(* Logix 5000 project; controller LeakTestAuto vendor 1 type 14 code 226 rev 37.11; software revision 37.01; part 5 of 12 *)
(* tags used below, declared in another part *)
   AOI_CTS1 : AOI_CTS_INSTRUMENT;
   AOI_CTS2 : AOI_CTS_INSTRUMENT;
   AOI_OP220_HomingSeq : AOI_Sequencer_x64;
   AOI_RobotPos : AOI_RobotPositions;
   AOI_SeqSteps : AOI_StandardSeqSteps;
   BarcodeScanner : udt_OutputStructure;
   Config_ConveyorHomeCounter : DINT;
   Config_ConveyorHomeCounterEnter : BOOL;
   Config_CylinderWaitTime : DINT;
   Config_CylinderWaitTimeEnter : BOOL;
   Config_MaxFailCount : DINT;
   Config_MaxFailCountEnter : BOOL;
   Conveyor : udt_OutputStructure;
   Conveyor_Seq : udt_SequenceStructure_X64;
   ConveyorHomeCounter : COUNTER;
   DryCycle_N1Ready : BOOL;
   DryCycle_N2Ready : BOOL;
   FailCount : COUNTER;
   HMI_CloseDisplay : DINT;
   HomingClearNestsBypass : BOOL;
   LeakTester1 : udt_OutputStructure;
   LeakTester2 : udt_OutputStructure;
   Mode_CapActuators : BOOL;
   Mode_CapCTS : BOOL;
   Mode_CapCylinders : BOOL;
   Mode_CapFail : BOOL;
   Mode_CapPass : BOOL;
   Mode_CapRobot : BOOL;
   Mode_CapShuffle : BOOL;
   Nest1Cylinder : udt_OutputStructure;
   Nest1Empty : BOOL;
   Nest1Ready : BOOL;
   Nest2Cylinder : udt_OutputStructure;
   Nest2Empty : BOOL;
   Nest2Ready : BOOL;
   ONS_CycleStop : BOOL;
   ONS_FailBinRemoved : BOOL;
   ONS_ManuMode : BOOL;
   OP220 : udt_Mode;
   OP220_HomingSeq : udt_SequenceStructure_X64;
   OP220_PartToPartCycleTMR : TIMER;
   OP220_Seq : udt_SequenceStructure_X64;
   RFIDScanner : udt_OutputStructure;
   Robot : udt_OutputStructure;
   RobotGripper : udt_OutputStructure;
   RobotInputs : udt_EpsonInputs;
   RobotOutputs : udt_EpsonOutputs;
   TON_FailChute : TIMER[10];
   TON_HMICloseDisplayDelay : TIMER;
   TON_Nest1DryCycleDryTest : TIMER;
   TON_Nest2DryCycleDryTest : TIMER;
   ConveyorPurgeCounter : DINT;   // Outfeed Coveyor Purge Counter
   HMI_PurgeCycleSP : DINT;   // HMI Purge Cycles Setpoint
   I_OP220_N3_CONVEYOR_CLEAT : ALIAS FOR Local:3:I.Pt13.Data;
   I_OP220_N3_DUT_PRE_NEST_1 : ALIAS FOR Local:3:I.Pt01.Data;
   I_OP220_N3_DUT_PRE_NEST_2 : ALIAS FOR Local:3:I.Pt02.Data;
   I_OP220_N3_MAIN_AIR_OK : ALIAS FOR Local:3:I.Pt07.Data;
   I_OP220_N3_NEST1_EXTEND : ALIAS FOR Local:3:I.Pt04.Data;
   I_OP220_N3_NEST1_HOME : ALIAS FOR Local:3:I.Pt03.Data;
   I_OP220_N3_NEST2_EXTEND : ALIAS FOR Local:3:I.Pt06.Data;
   I_OP220_N3_NEST2_HOME : ALIAS FOR Local:3:I.Pt05.Data;
   I_OP220_N3_REJECT_BIN_OK : ALIAS FOR Local:3:I.Pt09.Data;
   I_OP220_N3_REJECT_CHUTE_PART : ALIAS FOR Local:3:I.Pt10.Data;
   James_Dint : DINT;   // James Test Word
   O_OP220_N5_CONV_REV : ALIAS FOR Local:5:O.Pt11.Data;
   O_OP220_N5_EN_LT_BU : ALIAS FOR Local:5:O.Pt03.Data;
   O_OP220_N5_EN_LT_GN : ALIAS FOR Local:5:O.Pt00.Data;
   O_OP220_N5_EN_LT_RD : ALIAS FOR Local:5:O.Pt02.Data;
   O_OP220_N5_EN_LT_YE : ALIAS FOR Local:5:O.Pt01.Data;
   O_OP220_N5_EN_MAIN_AIR : ALIAS FOR Local:5:O.Pt04.Data;
   O_OP220_N5_EN_ROBOT_LATCHOFF : ALIAS FOR Local:5:O.Pt09.Data;
   OP220_ConsumedFromMain_PurgeModeEn : BOOL;
   OP220_Power : BOOL;
   PLC : AOI_PLC;
   Purge_Count_DN : BOOL;   // Purge Counter Completed
(* MainProgram, continued *)

ROUTINE R05_ModeControl   (* ladder *)
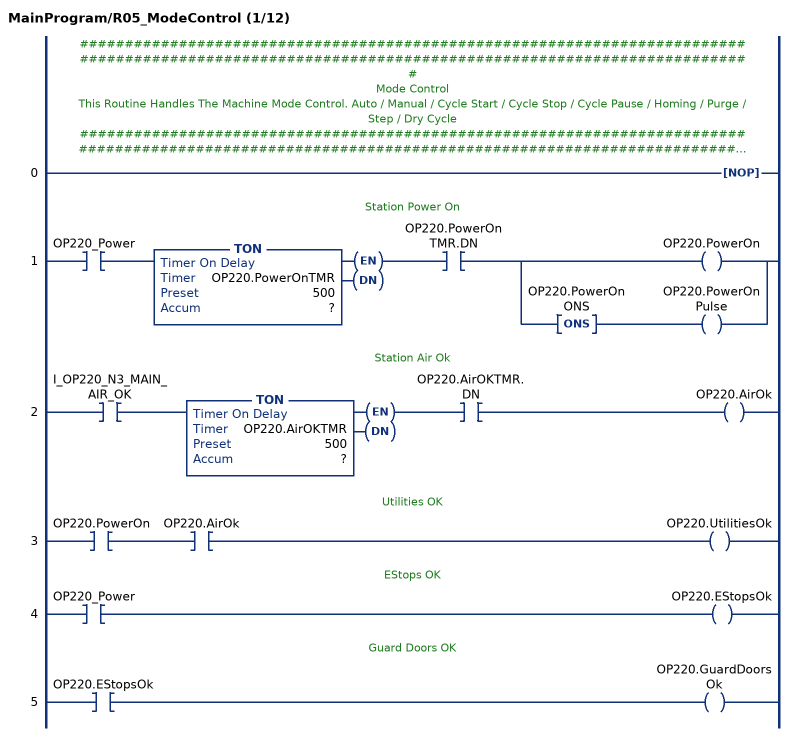
   // #####################################################################################################################################################
   // Mode Control
   // This Routine Handles The Machine Mode Control. Auto / Manual / Cycle Start / Cycle Stop / Cycle Pause / Homing / Purge / Step / Dry Cycle
   // #####################################################################################################################################################
   0: NOP();
   // Station Power On
   1: XIC(OP220_Power)TON(OP220.PowerOnTMR,?,?)XIC(OP220.PowerOnTMR.DN)[OTE(OP220.PowerOn) ,ONS(OP220.PowerOnONS) OTE(OP220.PowerOnPulse) ];
   // Station Air Ok
   2: XIC(I_OP220_N3_MAIN_AIR_OK)TON(OP220.AirOKTMR,?,?)XIC(OP220.AirOKTMR.DN)OTE(OP220.AirOk);
   // Utilities OK
   3: XIC(OP220.PowerOn)XIC(OP220.AirOk)OTE(OP220.UtilitiesOk);
   // EStops OK
   4: XIC(OP220_Power)OTE(OP220.EStopsOk);
   // Guard Doors OK
   5: XIC(OP220.EStopsOk)OTE(OP220.GuardDoorsOk);
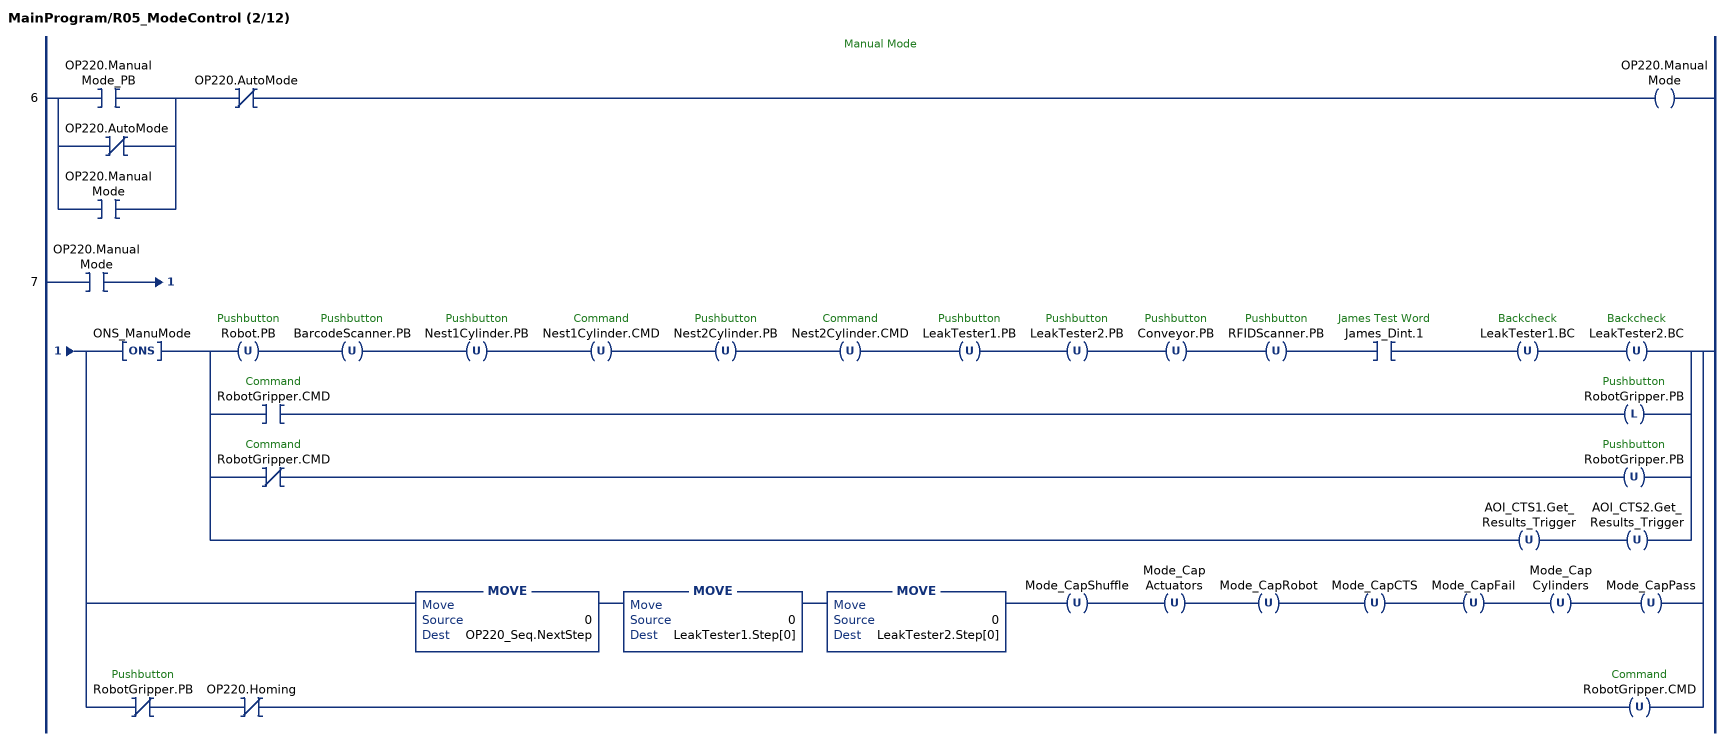
   // Manual Mode
   6: [XIC(OP220.ManualMode_PB) ,XIO(OP220.AutoMode) ,XIC(OP220.ManualMode) ]XIO(OP220.AutoMode)OTE(OP220.ManualMode);
   7: XIC(OP220.ManualMode)[ONS(ONS_ManuMode) [OTU(Robot.PB) OTU(BarcodeScanner.PB) OTU(Nest1Cylinder.PB) OTU(Nest1Cylinder.CMD) OTU(Nest2Cylinder.PB) OTU(Nest2Cylinder.CMD) OTU(LeakTester1.PB) OTU(LeakTester2.PB) OTU(Conveyor.PB) OTU(RFIDScanner.PB) XIC(James_Dint.1) OTU(LeakTester1.BC) OTU(LeakTester2.BC) ,XIC(RobotGripper.CMD) OTL(RobotGripper.PB) ,XIO(RobotGripper.CMD) OTU(RobotGripper.PB) ,OTU(AOI_CTS1.Get_Results_Trigger) OTU(AOI_CTS2.Get_Results_Trigger) ] ,MOVE(0,OP220_Seq.NextStep) MOVE(0,LeakTester1.Step[0]) MOVE(0,LeakTester2.Step[0]) OTU(Mode_CapShuffle) OTU(Mode_CapActuators) OTU(Mode_CapRobot) OTU(Mode_CapCTS) OTU(Mode_CapFail) OTU(Mode_CapCylinders) OTU(Mode_CapPass) ,XIO(RobotGripper.PB) XIO(OP220.Homing) OTU(RobotGripper.CMD) ];
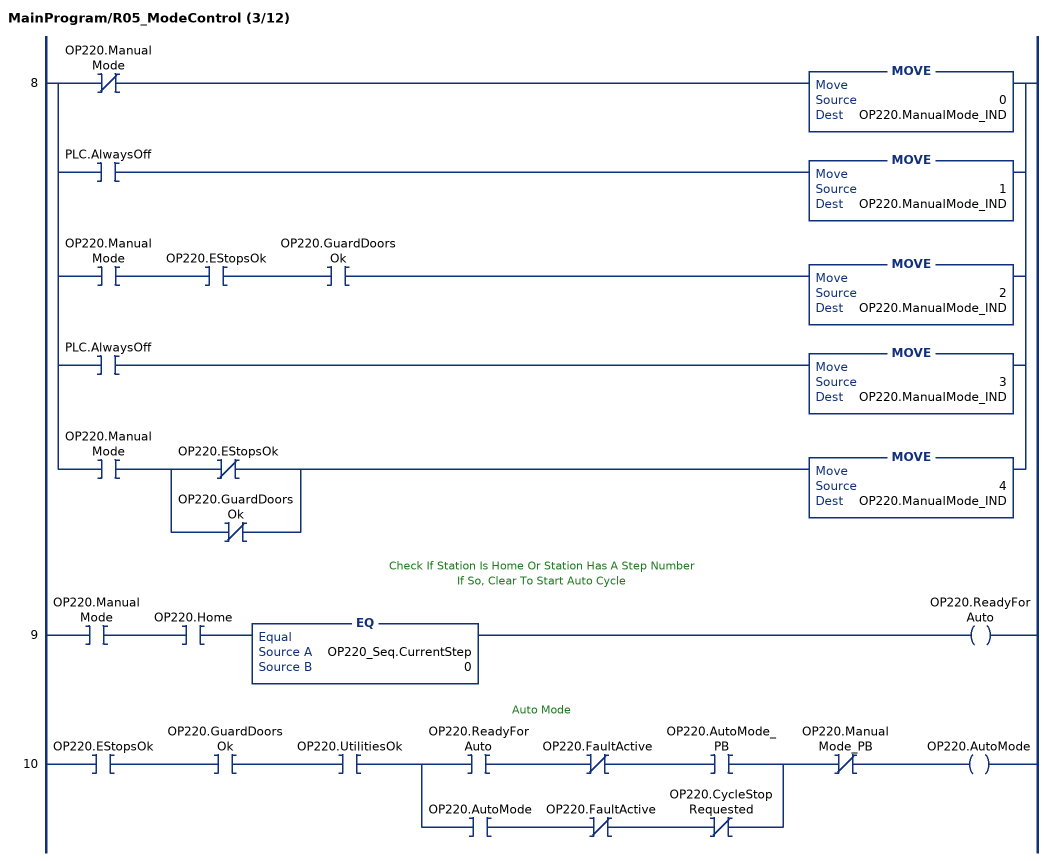
   8: [XIO(OP220.ManualMode) MOVE(0,OP220.ManualMode_IND) ,XIC(PLC.AlwaysOff) MOVE(1,OP220.ManualMode_IND) ,XIC(OP220.ManualMode) XIC(OP220.EStopsOk) XIC(OP220.GuardDoorsOk) MOVE(2,OP220.ManualMode_IND) ,XIC(PLC.AlwaysOff) MOVE(3,OP220.ManualMode_IND) ,XIC(OP220.ManualMode) [XIO(OP220.EStopsOk) ,XIO(OP220.GuardDoorsOk) ] MOVE(4,OP220.ManualMode_IND) ];
   // Check If Station Is Home Or Station Has A Step Number
   // If So, Clear To Start Auto Cycle
   9: XIC(OP220.ManualMode)XIC(OP220.Home)EQ(OP220_Seq.CurrentStep,0)OTE(OP220.ReadyForAuto);
   // Auto Mode
   10: XIC(OP220.EStopsOk)XIC(OP220.GuardDoorsOk)XIC(OP220.UtilitiesOk)[XIC(OP220.ReadyForAuto) XIO(OP220.FaultActive) XIC(OP220.AutoMode_PB) ,XIC(OP220.AutoMode) XIO(OP220.FaultActive) XIO(OP220.CycleStopRequested) ]XIO(OP220.ManualMode_PB)OTE(OP220.AutoMode);
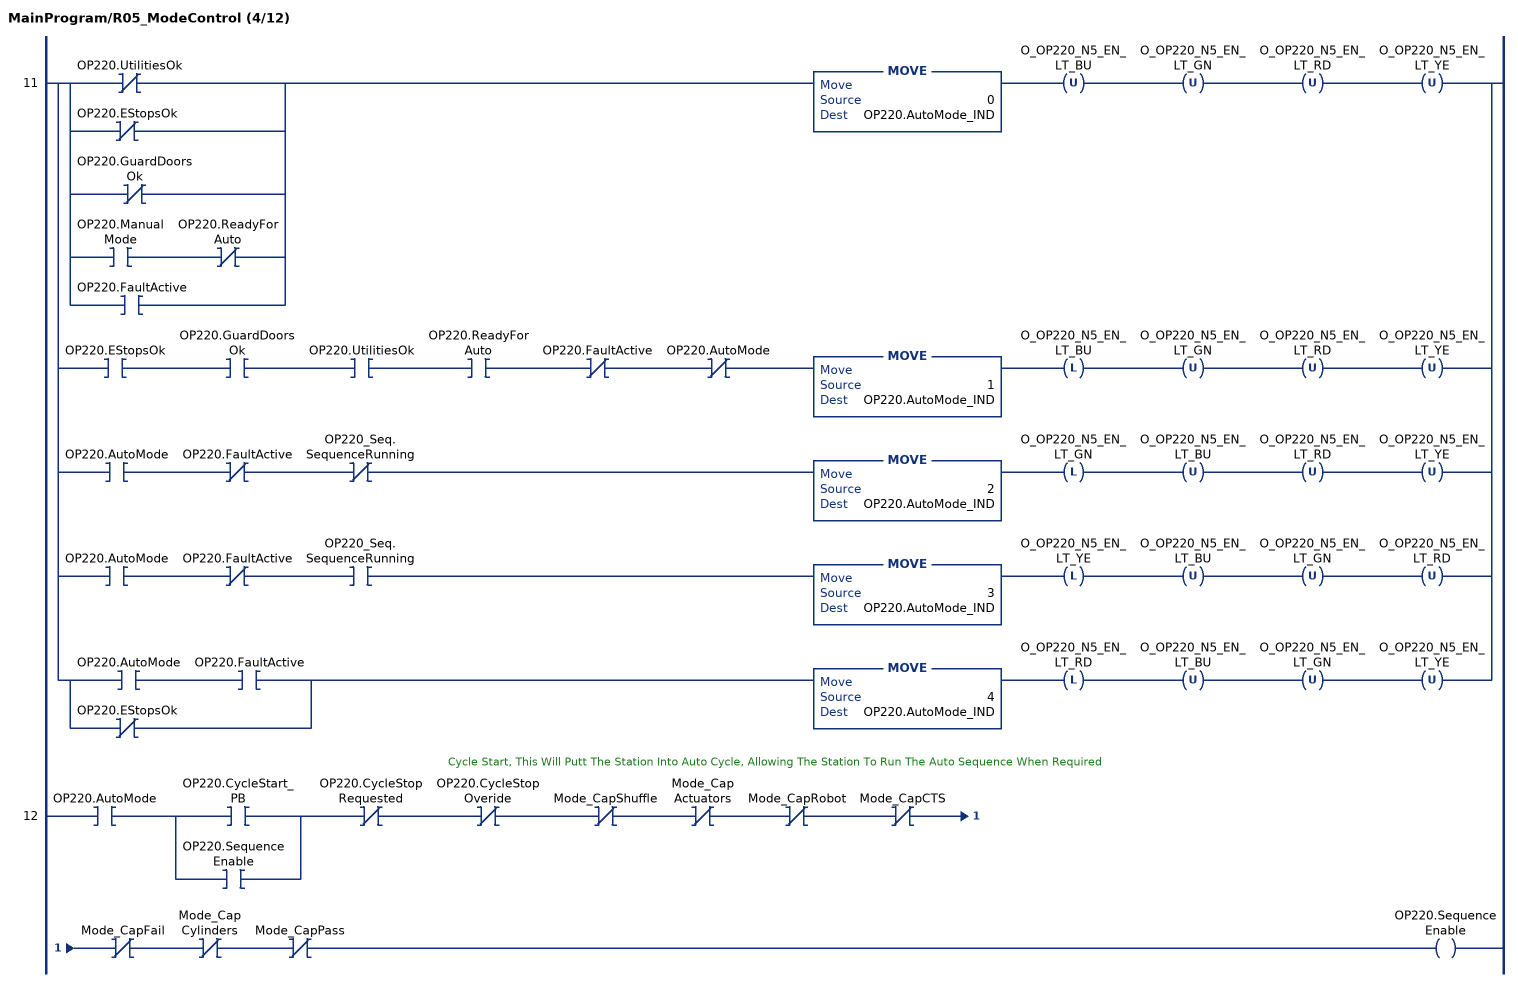
   11: [[XIO(OP220.UtilitiesOk) ,XIO(OP220.EStopsOk) ,XIO(OP220.GuardDoorsOk) ,XIC(OP220.ManualMode) XIO(OP220.ReadyForAuto) ,XIC(OP220.FaultActive) ] MOVE(0,OP220.AutoMode_IND) OTU(O_OP220_N5_EN_LT_BU) OTU(O_OP220_N5_EN_LT_GN) OTU(O_OP220_N5_EN_LT_RD) OTU(O_OP220_N5_EN_LT_YE) ,XIC(OP220.EStopsOk) XIC(OP220.GuardDoorsOk) XIC(OP220.UtilitiesOk) XIC(OP220.ReadyForAuto) XIO(OP220.FaultActive) XIO(OP220.AutoMode) MOVE(1,OP220.AutoMode_IND) OTL(O_OP220_N5_EN_LT_BU) OTU(O_OP220_N5_EN_LT_GN) OTU(O_OP220_N5_EN_LT_RD) OTU(O_OP220_N5_EN_LT_YE) ,XIC(OP220.AutoMode) XIO(OP220.FaultActive) XIO(OP220_Seq.SequenceRunning) MOVE(2,OP220.AutoMode_IND) OTL(O_OP220_N5_EN_LT_GN) OTU(O_OP220_N5_EN_LT_BU) OTU(O_OP220_N5_EN_LT_RD) OTU(O_OP220_N5_EN_LT_YE) ,XIC(OP220.AutoMode) XIO(OP220.FaultActive) XIC(OP220_Seq.SequenceRunning) MOVE(3,OP220.AutoMode_IND) OTL(O_OP220_N5_EN_LT_YE) OTU(O_OP220_N5_EN_LT_BU) OTU(O_OP220_N5_EN_LT_GN) OTU(O_OP220_N5_EN_LT_RD) ,[XIC(OP220.AutoMode) XIC(OP220.FaultActive) ,XIO(OP220.EStopsOk) ] MOVE(4,OP220.AutoMode_IND) OTL(O_OP220_N5_EN_LT_RD) OTU(O_OP220_N5_EN_LT_BU) OTU(O_OP220_N5_EN_LT_GN) OTU(O_OP220_N5_EN_LT_YE) ];
   // Cycle Start, This Will Putt The Station Into Auto Cycle, Allowing The Station To Run The Auto Sequence When Required
   12: XIC(OP220.AutoMode)[XIC(OP220.CycleStart_PB) ,XIC(OP220.SequenceEnable) ]XIO(OP220.CycleStopRequested)XIO(OP220.CycleStopOveride)XIO(Mode_CapShuffle)XIO(Mode_CapActuators)XIO(Mode_CapRobot)XIO(Mode_CapCTS)XIO(Mode_CapFail)XIO(Mode_CapCylinders)XIO(Mode_CapPass)OTE(OP220.SequenceEnable);
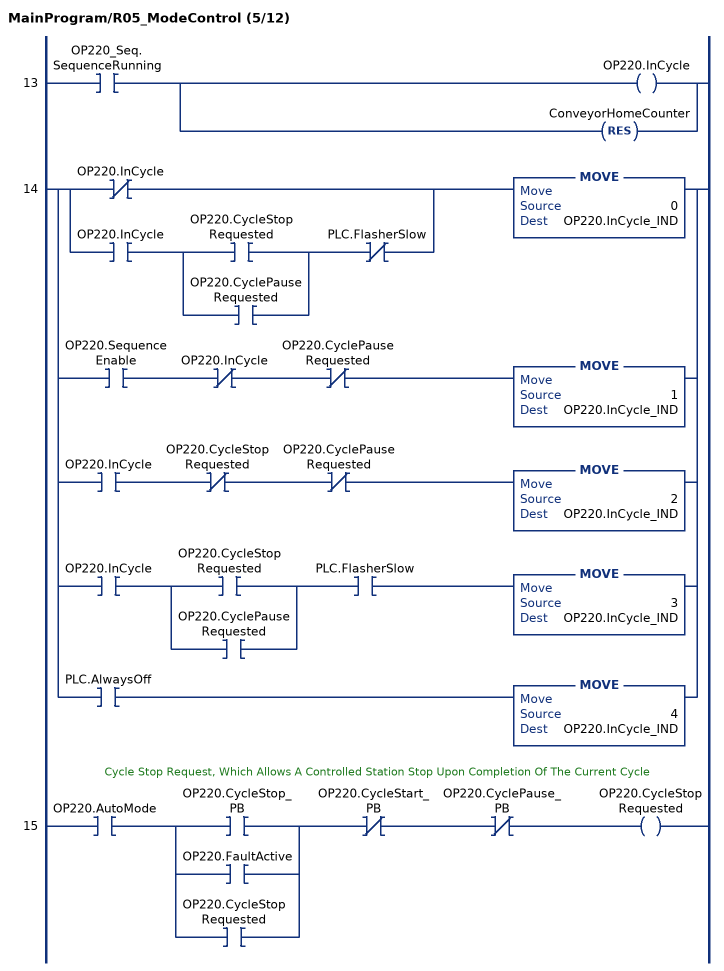
   13: XIC(OP220_Seq.SequenceRunning)[OTE(OP220.InCycle) ,RES(ConveyorHomeCounter) ];
   14: [[XIO(OP220.InCycle) ,XIC(OP220.InCycle) [XIC(OP220.CycleStopRequested) ,XIC(OP220.CyclePauseRequested) ] XIO(PLC.FlasherSlow) ] MOVE(0,OP220.InCycle_IND) ,XIC(OP220.SequenceEnable) XIO(OP220.InCycle) XIO(OP220.CyclePauseRequested) MOVE(1,OP220.InCycle_IND) ,XIC(OP220.InCycle) XIO(OP220.CycleStopRequested) XIO(OP220.CyclePauseRequested) MOVE(2,OP220.InCycle_IND) ,XIC(OP220.InCycle) [XIC(OP220.CycleStopRequested) ,XIC(OP220.CyclePauseRequested) ] XIC(PLC.FlasherSlow) MOVE(3,OP220.InCycle_IND) ,XIC(PLC.AlwaysOff) MOVE(4,OP220.InCycle_IND) ];
   // Cycle Stop Request, Which Allows A Controlled Station Stop Upon Completion Of The Current Cycle
   15: XIC(OP220.AutoMode)[XIC(OP220.CycleStop_PB) ,XIC(OP220.FaultActive) ,XIC(OP220.CycleStopRequested) ]XIO(OP220.CycleStart_PB)XIO(OP220.CyclePause_PB)OTE(OP220.CycleStopRequested);
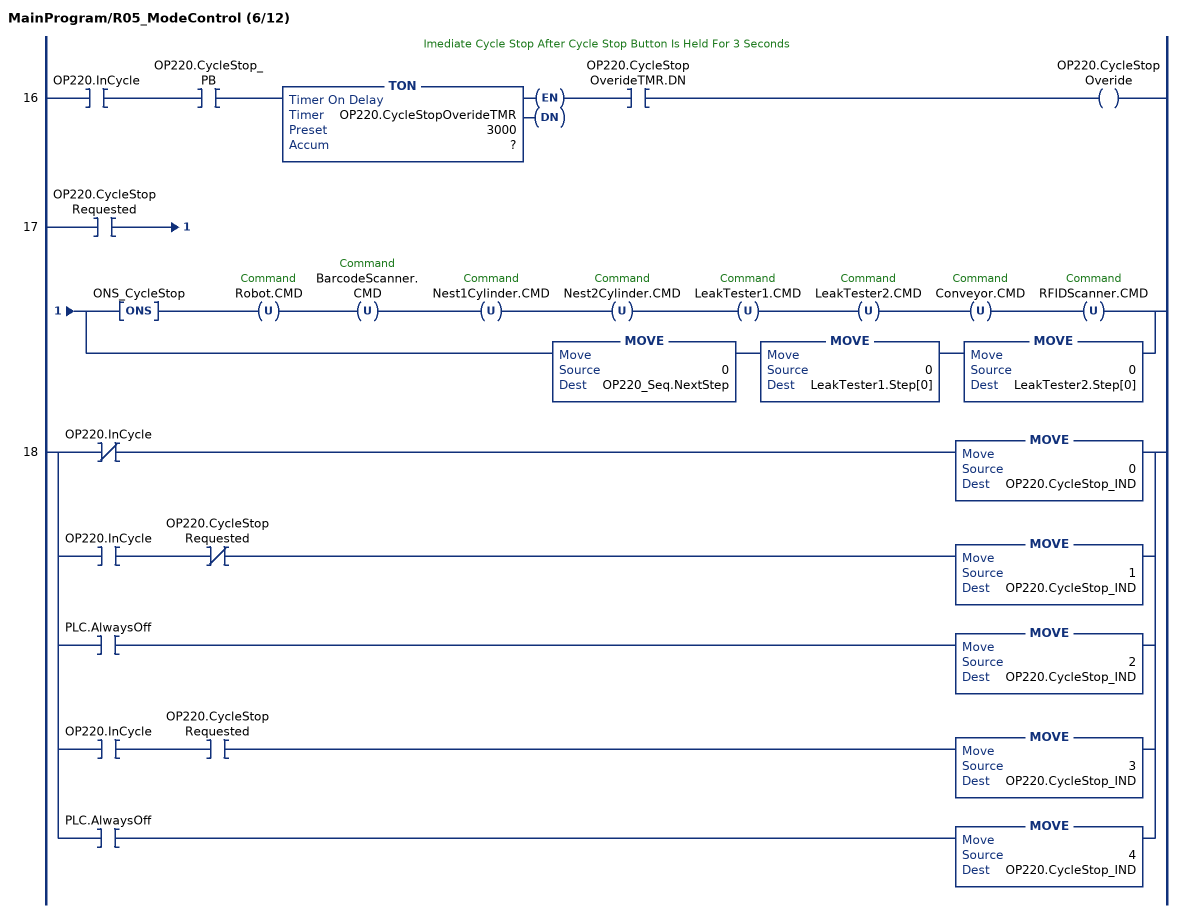
   // Imediate Cycle Stop After Cycle Stop Button Is Held For 3 Seconds
   16: XIC(OP220.InCycle)XIC(OP220.CycleStop_PB)TON(OP220.CycleStopOverideTMR,?,?)XIC(OP220.CycleStopOverideTMR.DN)OTE(OP220.CycleStopOveride);
   17: XIC(OP220.CycleStopRequested)[ONS(ONS_CycleStop) OTU(Robot.CMD) OTU(BarcodeScanner.CMD) OTU(Nest1Cylinder.CMD) OTU(Nest2Cylinder.CMD) OTU(LeakTester1.CMD) OTU(LeakTester2.CMD) OTU(Conveyor.CMD) OTU(RFIDScanner.CMD) ,MOVE(0,OP220_Seq.NextStep) MOVE(0,LeakTester1.Step[0]) MOVE(0,LeakTester2.Step[0]) ];
   18: [XIO(OP220.InCycle) MOVE(0,OP220.CycleStop_IND) ,XIC(OP220.InCycle) XIO(OP220.CycleStopRequested) MOVE(1,OP220.CycleStop_IND) ,XIC(PLC.AlwaysOff) MOVE(2,OP220.CycleStop_IND) ,XIC(OP220.InCycle) XIC(OP220.CycleStopRequested) MOVE(3,OP220.CycleStop_IND) ,XIC(PLC.AlwaysOff) MOVE(4,OP220.CycleStop_IND) ];
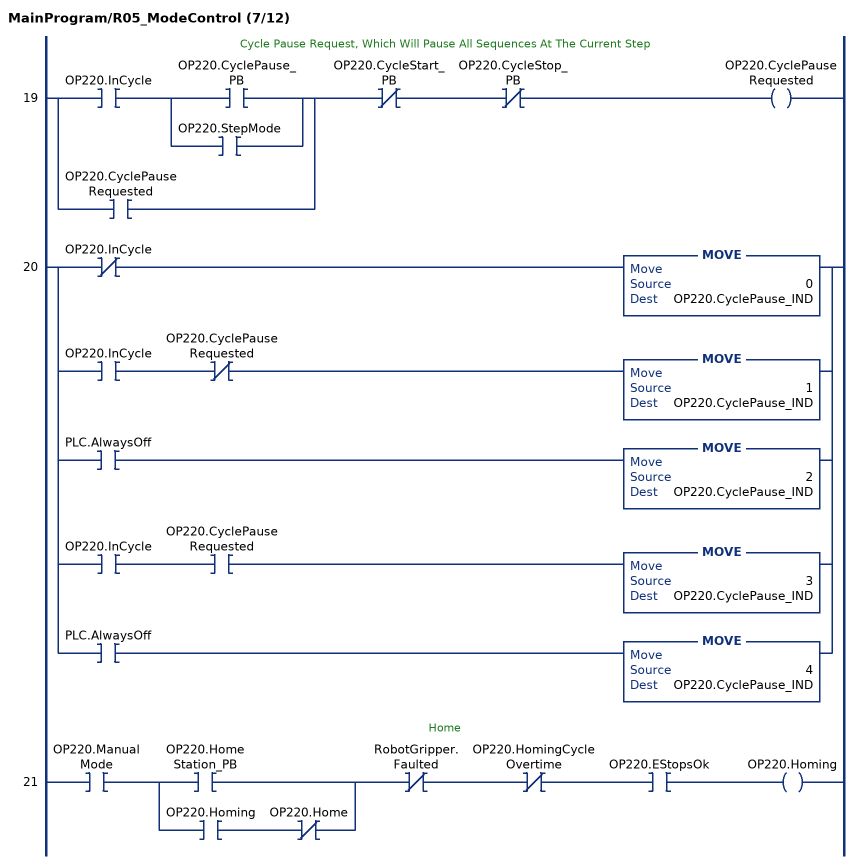
   // Cycle Pause Request, Which Will Pause All Sequences At The Current Step
   19: [XIC(OP220.InCycle) [XIC(OP220.CyclePause_PB) ,XIC(OP220.StepMode) ] ,XIC(OP220.CyclePauseRequested) ]XIO(OP220.CycleStart_PB)XIO(OP220.CycleStop_PB)OTE(OP220.CyclePauseRequested);
   20: [XIO(OP220.InCycle) MOVE(0,OP220.CyclePause_IND) ,XIC(OP220.InCycle) XIO(OP220.CyclePauseRequested) MOVE(1,OP220.CyclePause_IND) ,XIC(PLC.AlwaysOff) MOVE(2,OP220.CyclePause_IND) ,XIC(OP220.InCycle) XIC(OP220.CyclePauseRequested) MOVE(3,OP220.CyclePause_IND) ,XIC(PLC.AlwaysOff) MOVE(4,OP220.CyclePause_IND) ];
   // Home
   21: XIC(OP220.ManualMode)[XIC(OP220.HomeStation_PB) ,XIC(OP220.Homing) XIO(OP220.Home) ]XIO(RobotGripper.Faulted)XIO(OP220.HomingCycleOvertime)XIC(OP220.EStopsOk)OTE(OP220.Homing);
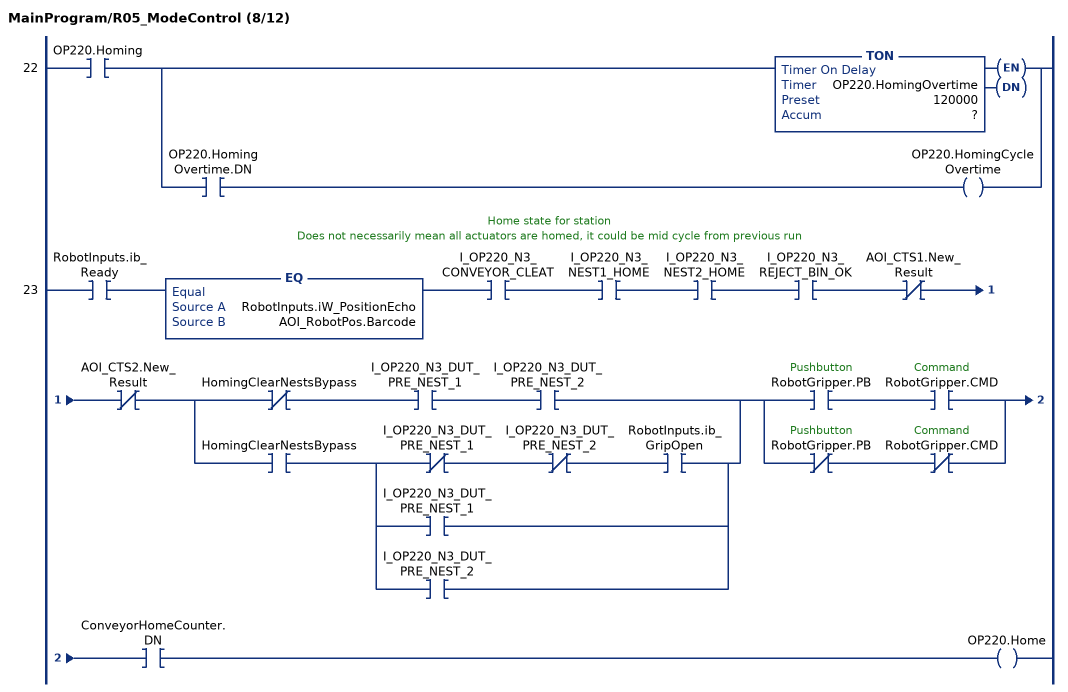
   22: XIC(OP220.Homing)[TON(OP220.HomingOvertime,?,?) ,XIC(OP220.HomingOvertime.DN) OTE(OP220.HomingCycleOvertime) ];
   // Home state for station
   // Does not necessarily mean all actuators are homed, it could be mid cycle from previous run
   23: XIC(RobotInputs.ib_Ready)EQ(RobotInputs.iW_PositionEcho,AOI_RobotPos.Barcode)XIC(I_OP220_N3_CONVEYOR_CLEAT)XIC(I_OP220_N3_NEST1_HOME)XIC(I_OP220_N3_NEST2_HOME)XIC(I_OP220_N3_REJECT_BIN_OK)XIO(AOI_CTS1.New_Result)XIO(AOI_CTS2.New_Result)[XIO(HomingClearNestsBypass) XIC(I_OP220_N3_DUT_PRE_NEST_1) XIC(I_OP220_N3_DUT_PRE_NEST_2) ,XIC(HomingClearNestsBypass) [XIO(I_OP220_N3_DUT_PRE_NEST_1) XIO(I_OP220_N3_DUT_PRE_NEST_2) XIC(RobotInputs.ib_GripOpen) ,XIC(I_OP220_N3_DUT_PRE_NEST_1) ,XIC(I_OP220_N3_DUT_PRE_NEST_2) ] ][XIC(RobotGripper.PB) XIC(RobotGripper.CMD) ,XIO(RobotGripper.PB) XIO(RobotGripper.CMD) ]XIC(ConveyorHomeCounter.DN)OTE(OP220.Home);
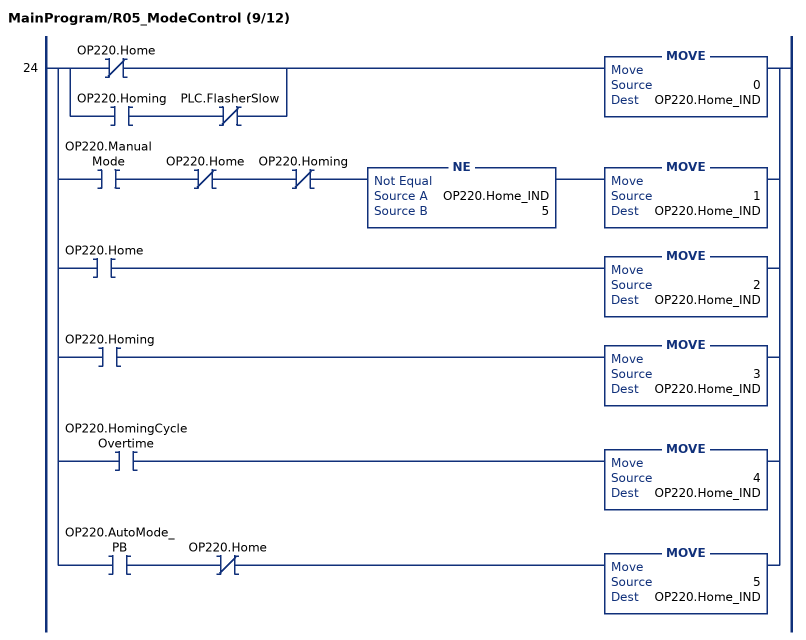
   24: [[XIO(OP220.Home) ,XIC(OP220.Homing) XIO(PLC.FlasherSlow) ] MOVE(0,OP220.Home_IND) ,XIC(OP220.ManualMode) XIO(OP220.Home) XIO(OP220.Homing) NE(OP220.Home_IND,5) MOVE(1,OP220.Home_IND) ,XIC(OP220.Home) MOVE(2,OP220.Home_IND) ,XIC(OP220.Homing) MOVE(3,OP220.Home_IND) ,XIC(OP220.HomingCycleOvertime) MOVE(4,OP220.Home_IND) ,XIC(OP220.AutoMode_PB) XIO(OP220.Home) MOVE(5,OP220.Home_IND) ];
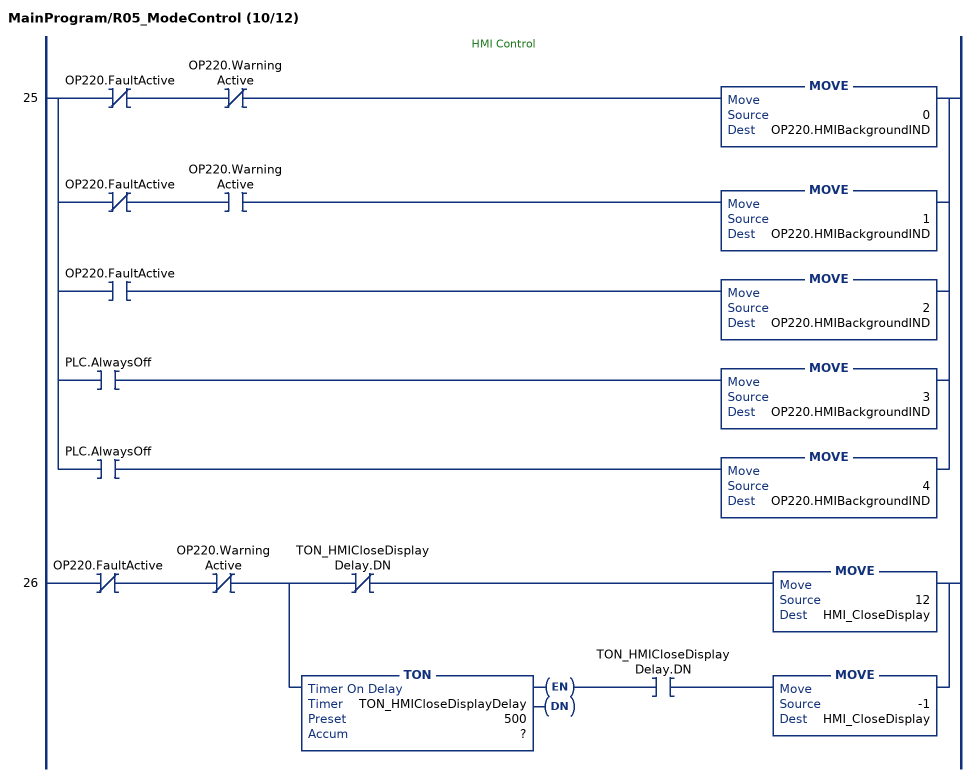
   // HMI Control
   25: [XIO(OP220.FaultActive) XIO(OP220.WarningActive) MOVE(0,OP220.HMIBackgroundIND) ,XIO(OP220.FaultActive) XIC(OP220.WarningActive) MOVE(1,OP220.HMIBackgroundIND) ,XIC(OP220.FaultActive) MOVE(2,OP220.HMIBackgroundIND) ,XIC(PLC.AlwaysOff) MOVE(3,OP220.HMIBackgroundIND) ,XIC(PLC.AlwaysOff) MOVE(4,OP220.HMIBackgroundIND) ];
   26: XIO(OP220.FaultActive)XIO(OP220.WarningActive)[XIO(TON_HMICloseDisplayDelay.DN) MOVE(12,HMI_CloseDisplay) ,TON(TON_HMICloseDisplayDelay,?,?) XIC(TON_HMICloseDisplayDelay.DN) MOVE(-1,HMI_CloseDisplay) ];
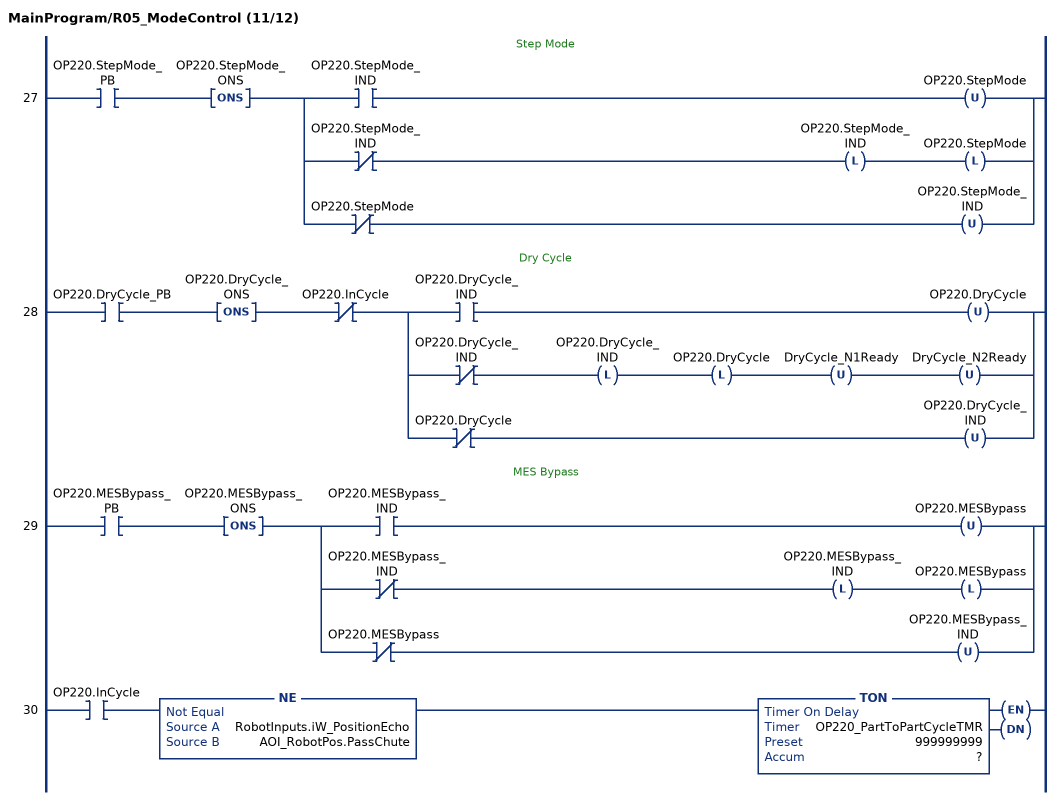
   // Step Mode
   27: XIC(OP220.StepMode_PB)ONS(OP220.StepMode_ONS)[XIC(OP220.StepMode_IND) OTU(OP220.StepMode) ,XIO(OP220.StepMode_IND) OTL(OP220.StepMode_IND) OTL(OP220.StepMode) ,XIO(OP220.StepMode) OTU(OP220.StepMode_IND) ];
   // Dry Cycle
   28: XIC(OP220.DryCycle_PB)ONS(OP220.DryCycle_ONS)XIO(OP220.InCycle)[XIC(OP220.DryCycle_IND) OTU(OP220.DryCycle) ,XIO(OP220.DryCycle_IND) OTL(OP220.DryCycle_IND) OTL(OP220.DryCycle) OTU(DryCycle_N1Ready) OTU(DryCycle_N2Ready) ,XIO(OP220.DryCycle) OTU(OP220.DryCycle_IND) ];
   // MES Bypass
   29: XIC(OP220.MESBypass_PB)ONS(OP220.MESBypass_ONS)[XIC(OP220.MESBypass_IND) OTU(OP220.MESBypass) ,XIO(OP220.MESBypass_IND) OTL(OP220.MESBypass_IND) OTL(OP220.MESBypass) ,XIO(OP220.MESBypass) OTU(OP220.MESBypass_IND) ];
   30: XIC(OP220.InCycle)NE(RobotInputs.iW_PositionEcho,AOI_RobotPos.PassChute)TON(OP220_PartToPartCycleTMR,?,?);
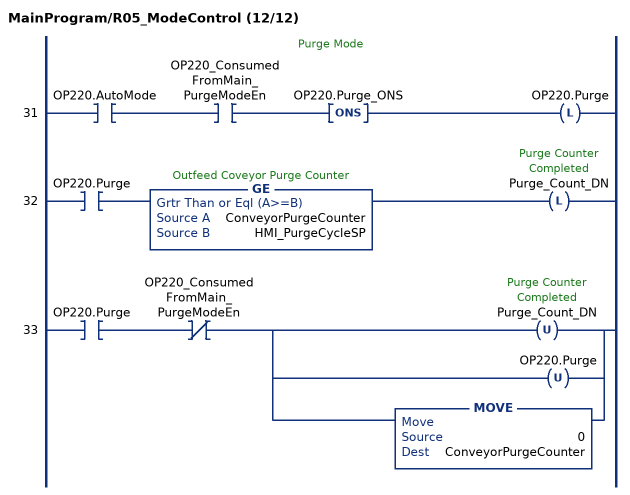
   // Purge Mode
   31: XIC(OP220.AutoMode)XIC(OP220_ConsumedFromMain_PurgeModeEn)ONS(OP220.Purge_ONS)OTL(OP220.Purge);
   32: XIC(OP220.Purge)GE(ConveyorPurgeCounter,HMI_PurgeCycleSP)OTL(Purge_Count_DN);
   33: XIC(OP220.Purge)XIO(OP220_ConsumedFromMain_PurgeModeEn)[OTU(Purge_Count_DN) ,OTU(OP220.Purge) ,MOVE(0,ConveyorPurgeCounter) ];
END_ROUTINE

ROUTINE R06_IOControl   (* ladder *)
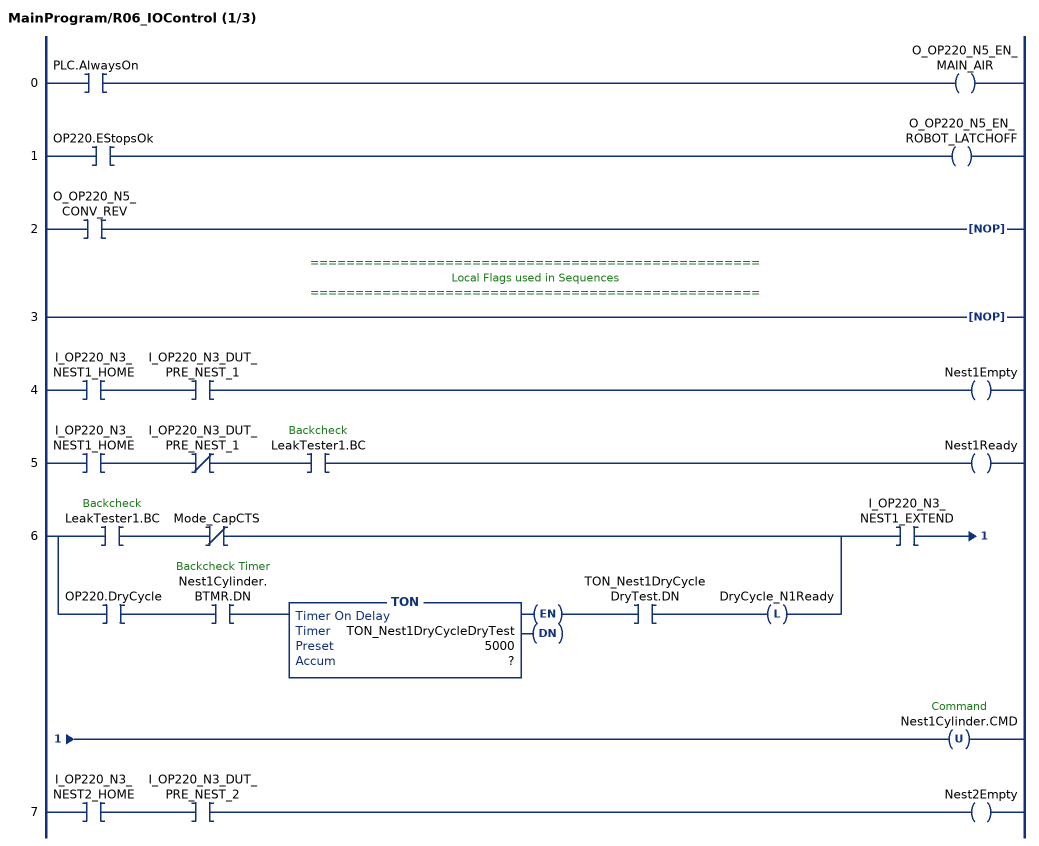
   0: XIC(PLC.AlwaysOn)OTE(O_OP220_N5_EN_MAIN_AIR);
   1: XIC(OP220.EStopsOk)OTE(O_OP220_N5_EN_ROBOT_LATCHOFF);
   2: XIC(O_OP220_N5_CONV_REV)NOP();
   // ==================================================
   // Local Flags used in Sequences
   // ==================================================
   3: NOP();
   4: XIC(I_OP220_N3_NEST1_HOME)XIC(I_OP220_N3_DUT_PRE_NEST_1)OTE(Nest1Empty);
   5: XIC(I_OP220_N3_NEST1_HOME)XIO(I_OP220_N3_DUT_PRE_NEST_1)XIC(LeakTester1.BC)OTE(Nest1Ready);
   6: [XIC(LeakTester1.BC) XIO(Mode_CapCTS) ,XIC(OP220.DryCycle) XIC(Nest1Cylinder.BTMR.DN) TON(TON_Nest1DryCycleDryTest,?,?) XIC(TON_Nest1DryCycleDryTest.DN) OTL(DryCycle_N1Ready) ]XIC(I_OP220_N3_NEST1_EXTEND)OTU(Nest1Cylinder.CMD);
   7: XIC(I_OP220_N3_NEST2_HOME)XIC(I_OP220_N3_DUT_PRE_NEST_2)OTE(Nest2Empty);
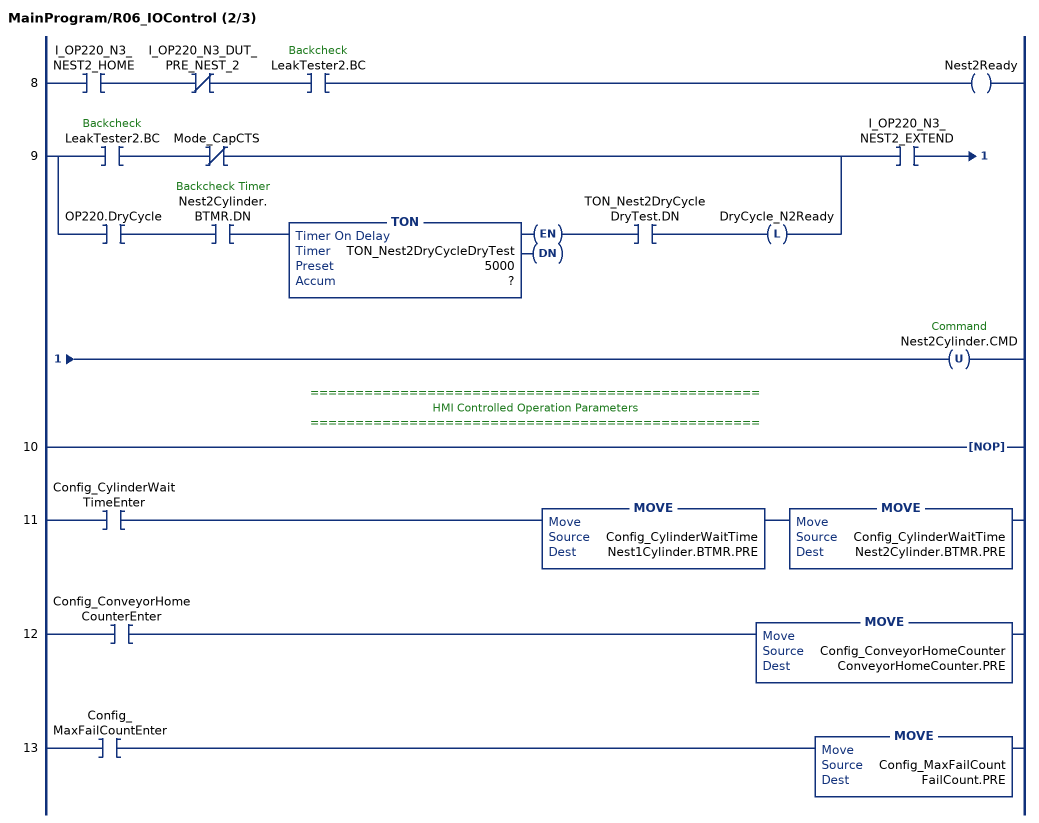
   8: XIC(I_OP220_N3_NEST2_HOME)XIO(I_OP220_N3_DUT_PRE_NEST_2)XIC(LeakTester2.BC)OTE(Nest2Ready);
   9: [XIC(LeakTester2.BC) XIO(Mode_CapCTS) ,XIC(OP220.DryCycle) XIC(Nest2Cylinder.BTMR.DN) TON(TON_Nest2DryCycleDryTest,?,?) XIC(TON_Nest2DryCycleDryTest.DN) OTL(DryCycle_N2Ready) ]XIC(I_OP220_N3_NEST2_EXTEND)OTU(Nest2Cylinder.CMD);
   // ==================================================
   // HMI Controlled Operation Parameters
   // ==================================================
   10: NOP();
   11: XIC(Config_CylinderWaitTimeEnter)MOVE(Config_CylinderWaitTime,Nest1Cylinder.BTMR.PRE)MOVE(Config_CylinderWaitTime,Nest2Cylinder.BTMR.PRE);
   12: XIC(Config_ConveyorHomeCounterEnter)MOVE(Config_ConveyorHomeCounter,ConveyorHomeCounter.PRE);
   13: XIC(Config_MaxFailCountEnter)MOVE(Config_MaxFailCount,FailCount.PRE);
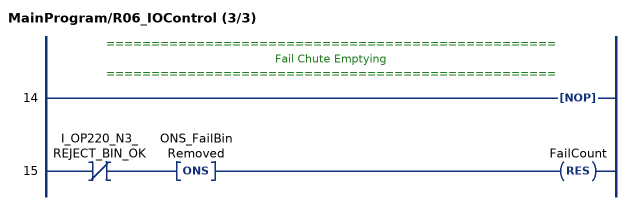
   // ==================================================
   // Fail Chute Emptying
   // ==================================================
   14: NOP();
   15: XIO(I_OP220_N3_REJECT_BIN_OK)ONS(ONS_FailBinRemoved)RES(FailCount);
END_ROUTINE

ROUTINE R09_Homing   (* ladder *)
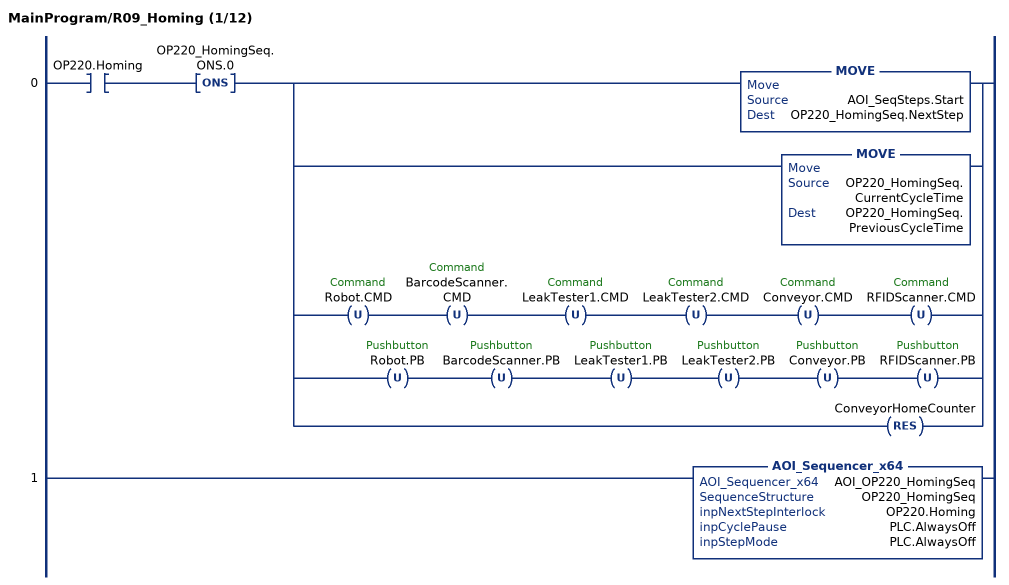
   0: XIC(OP220.Homing)ONS(OP220_HomingSeq.ONS.0)[MOVE(AOI_SeqSteps.Start,OP220_HomingSeq.NextStep) ,MOVE(OP220_HomingSeq.CurrentCycleTime,OP220_HomingSeq.PreviousCycleTime) ,OTU(Robot.CMD) OTU(BarcodeScanner.CMD) OTU(LeakTester1.CMD) OTU(LeakTester2.CMD) OTU(Conveyor.CMD) OTU(RFIDScanner.CMD) ,OTU(Robot.PB) OTU(BarcodeScanner.PB) OTU(LeakTester1.PB) OTU(LeakTester2.PB) OTU(Conveyor.PB) OTU(RFIDScanner.PB) ,RES(ConveyorHomeCounter) ];
   1: AOI_Sequencer_x64(AOI_OP220_HomingSeq,OP220_HomingSeq,OP220.Homing,PLC.AlwaysOff,PLC.AlwaysOff);
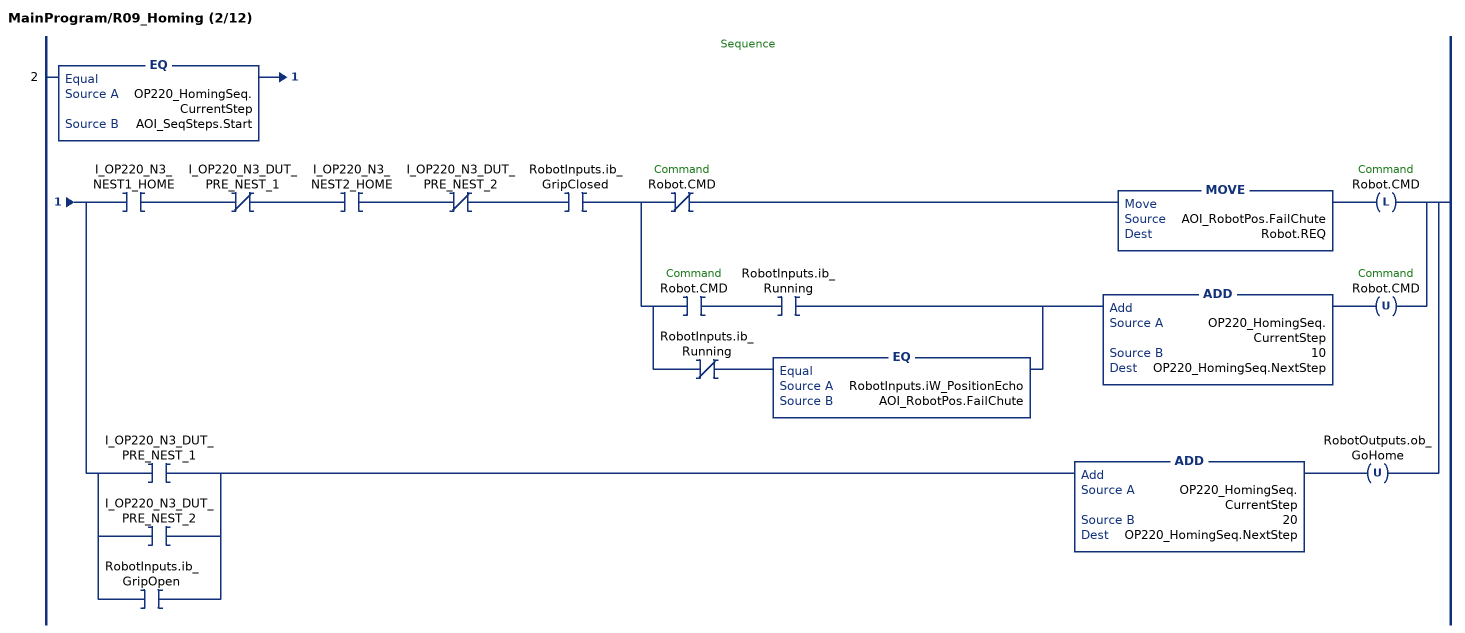
   // Sequence
   2: EQ(OP220_HomingSeq.CurrentStep,AOI_SeqSteps.Start)[XIC(I_OP220_N3_NEST1_HOME) XIO(I_OP220_N3_DUT_PRE_NEST_1) XIC(I_OP220_N3_NEST2_HOME) XIO(I_OP220_N3_DUT_PRE_NEST_2) XIC(RobotInputs.ib_GripClosed) [XIO(Robot.CMD) MOVE(AOI_RobotPos.FailChute,Robot.REQ) OTL(Robot.CMD) ,[XIC(Robot.CMD) XIC(RobotInputs.ib_Running) ,XIO(RobotInputs.ib_Running) EQ(RobotInputs.iW_PositionEcho,AOI_RobotPos.FailChute) ] ADD(OP220_HomingSeq.CurrentStep,10,OP220_HomingSeq.NextStep) OTU(Robot.CMD) ] ,[XIC(I_OP220_N3_DUT_PRE_NEST_1) ,XIC(I_OP220_N3_DUT_PRE_NEST_2) ,XIC(RobotInputs.ib_GripOpen) ] ADD(OP220_HomingSeq.CurrentStep,20,OP220_HomingSeq.NextStep) OTU(RobotOutputs.ob_GoHome) ];
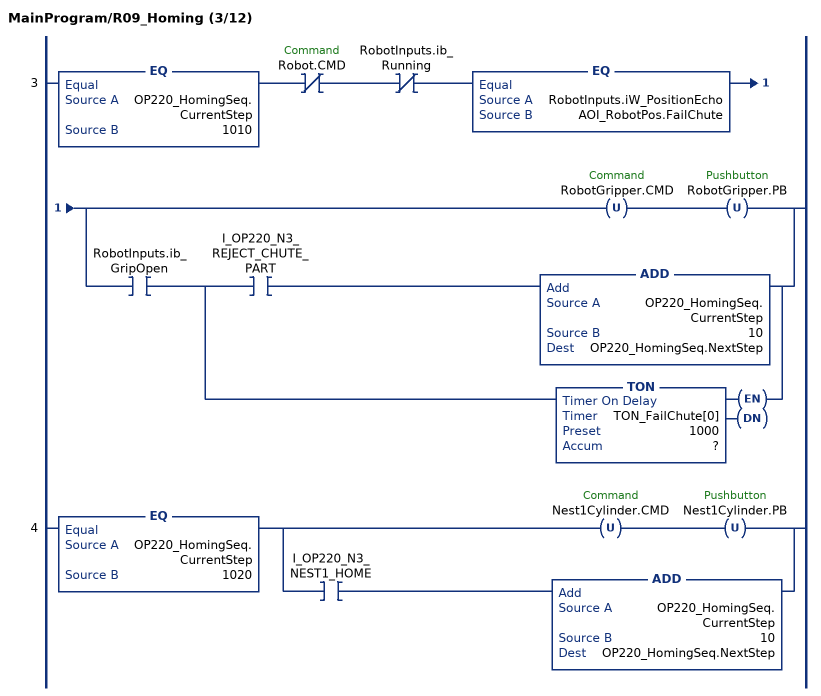
   3: EQ(OP220_HomingSeq.CurrentStep,1010)XIO(Robot.CMD)XIO(RobotInputs.ib_Running)EQ(RobotInputs.iW_PositionEcho,AOI_RobotPos.FailChute)[OTU(RobotGripper.CMD) OTU(RobotGripper.PB) ,XIC(RobotInputs.ib_GripOpen) [XIC(I_OP220_N3_REJECT_CHUTE_PART) ADD(OP220_HomingSeq.CurrentStep,10,OP220_HomingSeq.NextStep) ,TON(TON_FailChute[0],?,?) ] ];
   4: EQ(OP220_HomingSeq.CurrentStep,1020)[OTU(Nest1Cylinder.CMD) OTU(Nest1Cylinder.PB) ,XIC(I_OP220_N3_NEST1_HOME) ADD(OP220_HomingSeq.CurrentStep,10,OP220_HomingSeq.NextStep) ];
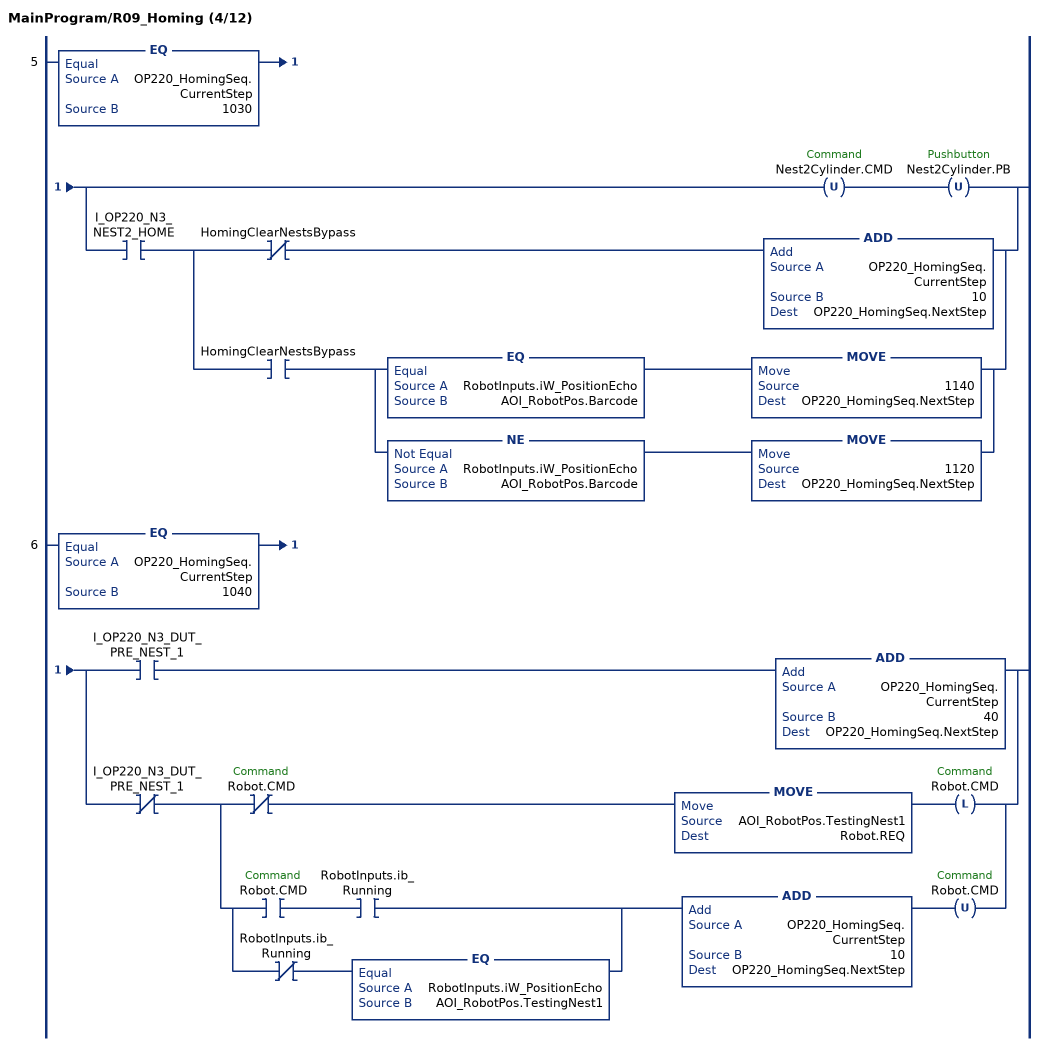
   5: EQ(OP220_HomingSeq.CurrentStep,1030)[OTU(Nest2Cylinder.CMD) OTU(Nest2Cylinder.PB) ,XIC(I_OP220_N3_NEST2_HOME) [XIO(HomingClearNestsBypass) ADD(OP220_HomingSeq.CurrentStep,10,OP220_HomingSeq.NextStep) ,XIC(HomingClearNestsBypass) [EQ(RobotInputs.iW_PositionEcho,AOI_RobotPos.Barcode) MOVE(1140,OP220_HomingSeq.NextStep) ,NE(RobotInputs.iW_PositionEcho,AOI_RobotPos.Barcode) MOVE(1120,OP220_HomingSeq.NextStep) ] ] ];
   6: EQ(OP220_HomingSeq.CurrentStep,1040)[XIC(I_OP220_N3_DUT_PRE_NEST_1) ADD(OP220_HomingSeq.CurrentStep,40,OP220_HomingSeq.NextStep) ,XIO(I_OP220_N3_DUT_PRE_NEST_1) [XIO(Robot.CMD) MOVE(AOI_RobotPos.TestingNest1,Robot.REQ) OTL(Robot.CMD) ,[XIC(Robot.CMD) XIC(RobotInputs.ib_Running) ,XIO(RobotInputs.ib_Running) EQ(RobotInputs.iW_PositionEcho,AOI_RobotPos.TestingNest1) ] ADD(OP220_HomingSeq.CurrentStep,10,OP220_HomingSeq.NextStep) OTU(Robot.CMD) ] ];
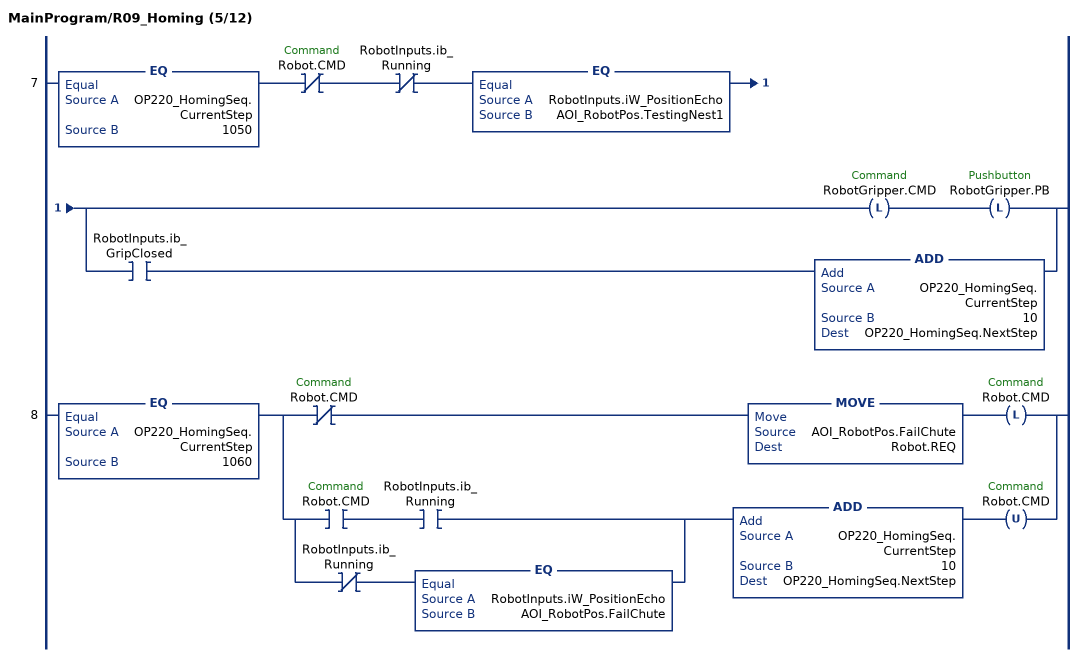
   7: EQ(OP220_HomingSeq.CurrentStep,1050)XIO(Robot.CMD)XIO(RobotInputs.ib_Running)EQ(RobotInputs.iW_PositionEcho,AOI_RobotPos.TestingNest1)[OTL(RobotGripper.CMD) OTL(RobotGripper.PB) ,XIC(RobotInputs.ib_GripClosed) ADD(OP220_HomingSeq.CurrentStep,10,OP220_HomingSeq.NextStep) ];
   8: EQ(OP220_HomingSeq.CurrentStep,1060)[XIO(Robot.CMD) MOVE(AOI_RobotPos.FailChute,Robot.REQ) OTL(Robot.CMD) ,[XIC(Robot.CMD) XIC(RobotInputs.ib_Running) ,XIO(RobotInputs.ib_Running) EQ(RobotInputs.iW_PositionEcho,AOI_RobotPos.FailChute) ] ADD(OP220_HomingSeq.CurrentStep,10,OP220_HomingSeq.NextStep) OTU(Robot.CMD) ];
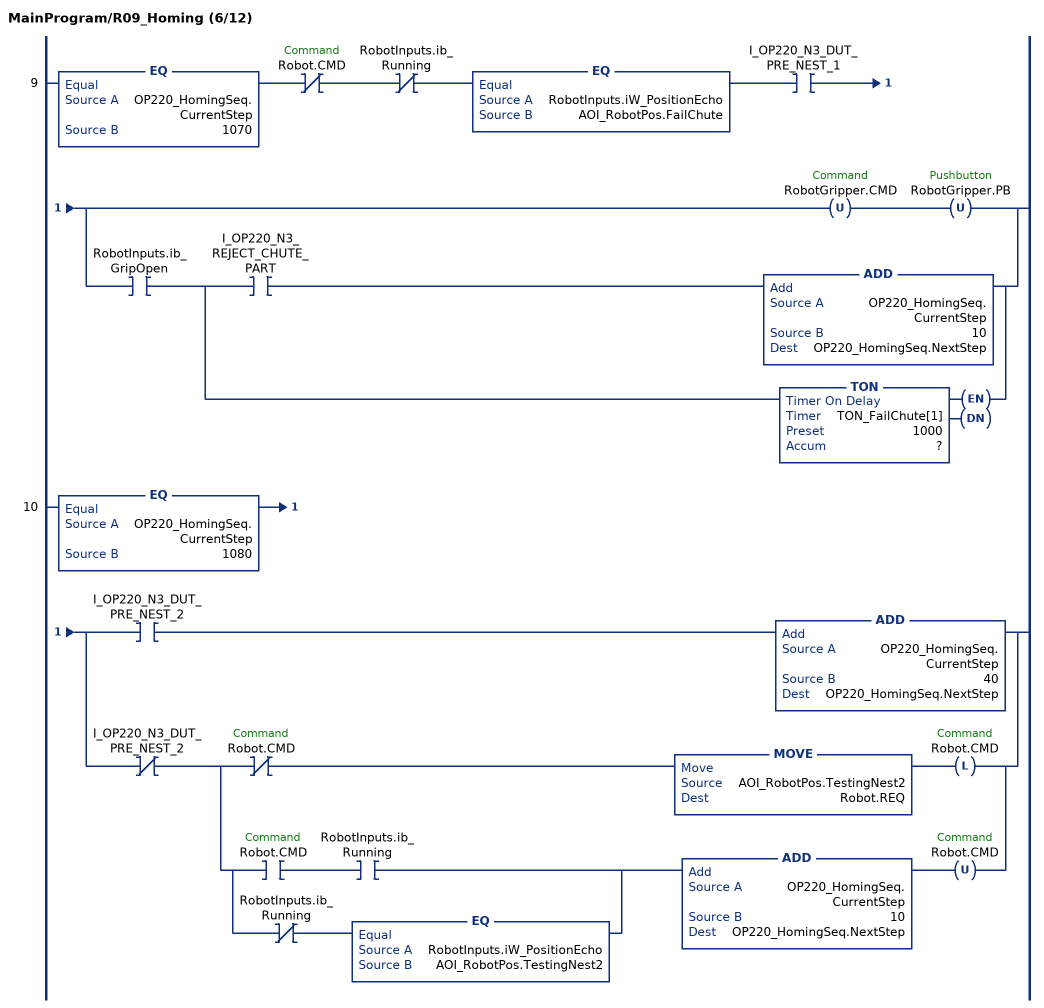
   9: EQ(OP220_HomingSeq.CurrentStep,1070)XIO(Robot.CMD)XIO(RobotInputs.ib_Running)EQ(RobotInputs.iW_PositionEcho,AOI_RobotPos.FailChute)XIC(I_OP220_N3_DUT_PRE_NEST_1)[OTU(RobotGripper.CMD) OTU(RobotGripper.PB) ,XIC(RobotInputs.ib_GripOpen) [XIC(I_OP220_N3_REJECT_CHUTE_PART) ADD(OP220_HomingSeq.CurrentStep,10,OP220_HomingSeq.NextStep) ,TON(TON_FailChute[1],?,?) ] ];
   10: EQ(OP220_HomingSeq.CurrentStep,1080)[XIC(I_OP220_N3_DUT_PRE_NEST_2) ADD(OP220_HomingSeq.CurrentStep,40,OP220_HomingSeq.NextStep) ,XIO(I_OP220_N3_DUT_PRE_NEST_2) [XIO(Robot.CMD) MOVE(AOI_RobotPos.TestingNest2,Robot.REQ) OTL(Robot.CMD) ,[XIC(Robot.CMD) XIC(RobotInputs.ib_Running) ,XIO(RobotInputs.ib_Running) EQ(RobotInputs.iW_PositionEcho,AOI_RobotPos.TestingNest2) ] ADD(OP220_HomingSeq.CurrentStep,10,OP220_HomingSeq.NextStep) OTU(Robot.CMD) ] ];
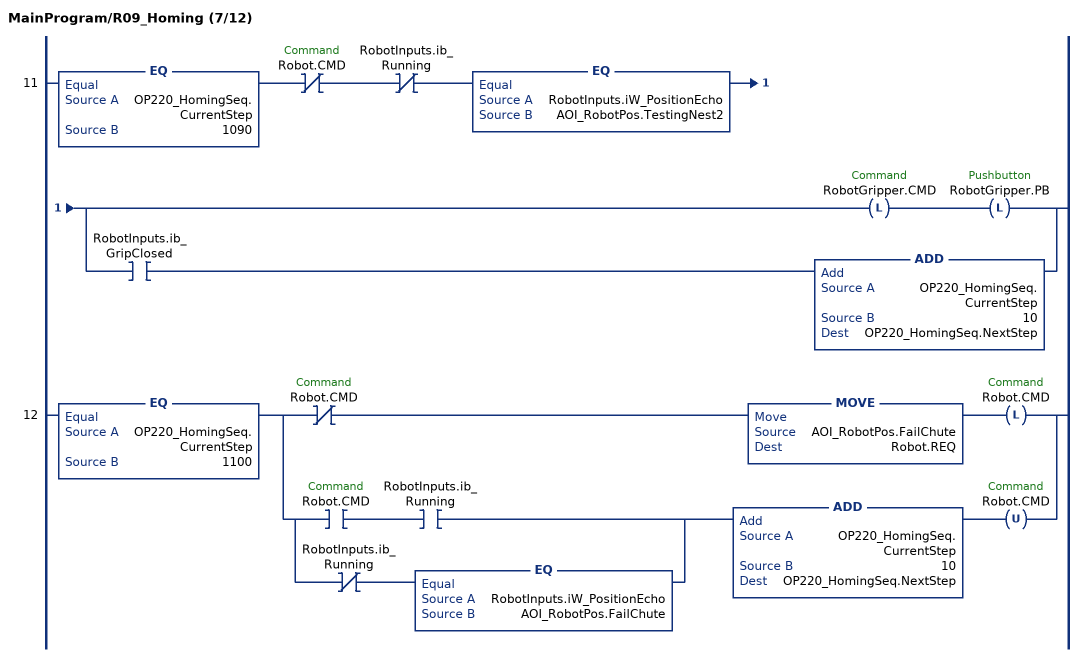
   11: EQ(OP220_HomingSeq.CurrentStep,1090)XIO(Robot.CMD)XIO(RobotInputs.ib_Running)EQ(RobotInputs.iW_PositionEcho,AOI_RobotPos.TestingNest2)[OTL(RobotGripper.CMD) OTL(RobotGripper.PB) ,XIC(RobotInputs.ib_GripClosed) ADD(OP220_HomingSeq.CurrentStep,10,OP220_HomingSeq.NextStep) ];
   12: EQ(OP220_HomingSeq.CurrentStep,1100)[XIO(Robot.CMD) MOVE(AOI_RobotPos.FailChute,Robot.REQ) OTL(Robot.CMD) ,[XIC(Robot.CMD) XIC(RobotInputs.ib_Running) ,XIO(RobotInputs.ib_Running) EQ(RobotInputs.iW_PositionEcho,AOI_RobotPos.FailChute) ] ADD(OP220_HomingSeq.CurrentStep,10,OP220_HomingSeq.NextStep) OTU(Robot.CMD) ];
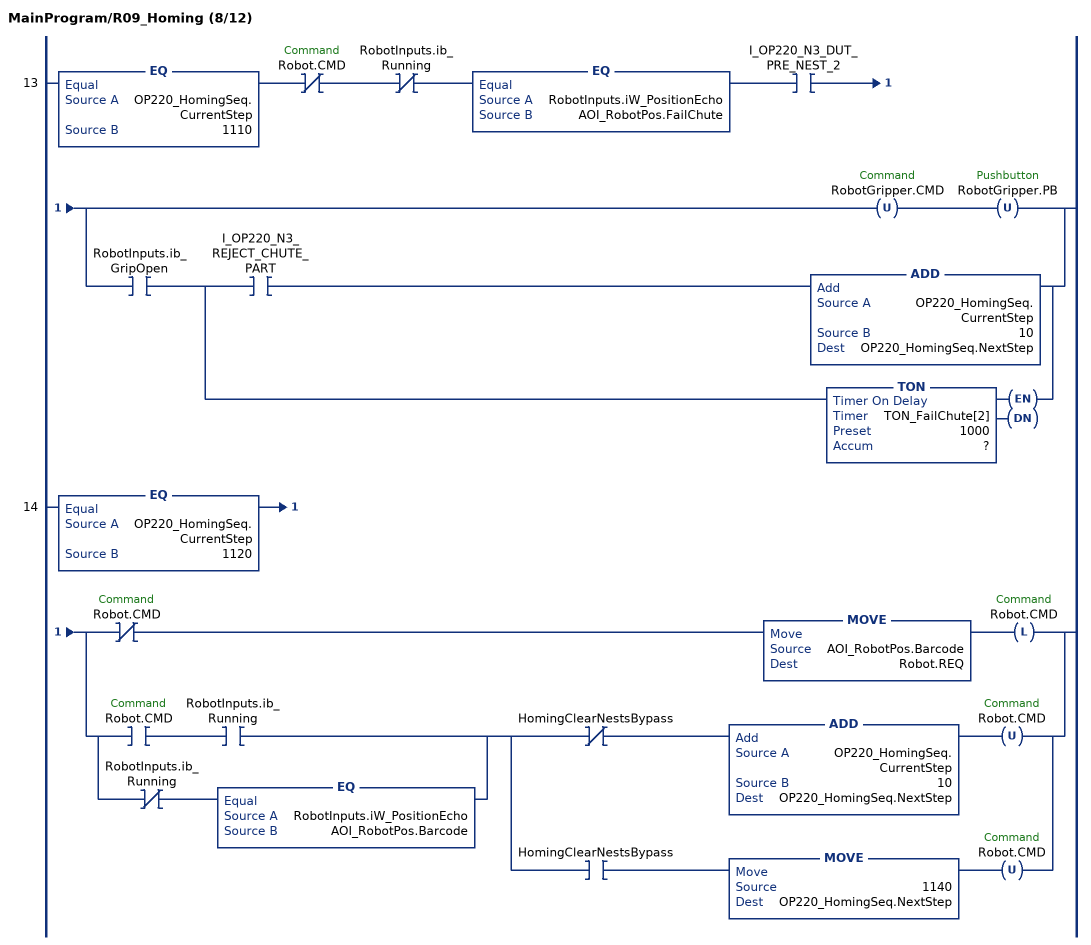
   13: EQ(OP220_HomingSeq.CurrentStep,1110)XIO(Robot.CMD)XIO(RobotInputs.ib_Running)EQ(RobotInputs.iW_PositionEcho,AOI_RobotPos.FailChute)XIC(I_OP220_N3_DUT_PRE_NEST_2)[OTU(RobotGripper.CMD) OTU(RobotGripper.PB) ,XIC(RobotInputs.ib_GripOpen) [XIC(I_OP220_N3_REJECT_CHUTE_PART) ADD(OP220_HomingSeq.CurrentStep,10,OP220_HomingSeq.NextStep) ,TON(TON_FailChute[2],?,?) ] ];
   14: EQ(OP220_HomingSeq.CurrentStep,1120)[XIO(Robot.CMD) MOVE(AOI_RobotPos.Barcode,Robot.REQ) OTL(Robot.CMD) ,[XIC(Robot.CMD) XIC(RobotInputs.ib_Running) ,XIO(RobotInputs.ib_Running) EQ(RobotInputs.iW_PositionEcho,AOI_RobotPos.Barcode) ] [XIO(HomingClearNestsBypass) ADD(OP220_HomingSeq.CurrentStep,10,OP220_HomingSeq.NextStep) OTU(Robot.CMD) ,XIC(HomingClearNestsBypass) MOVE(1140,OP220_HomingSeq.NextStep) OTU(Robot.CMD) ] ];
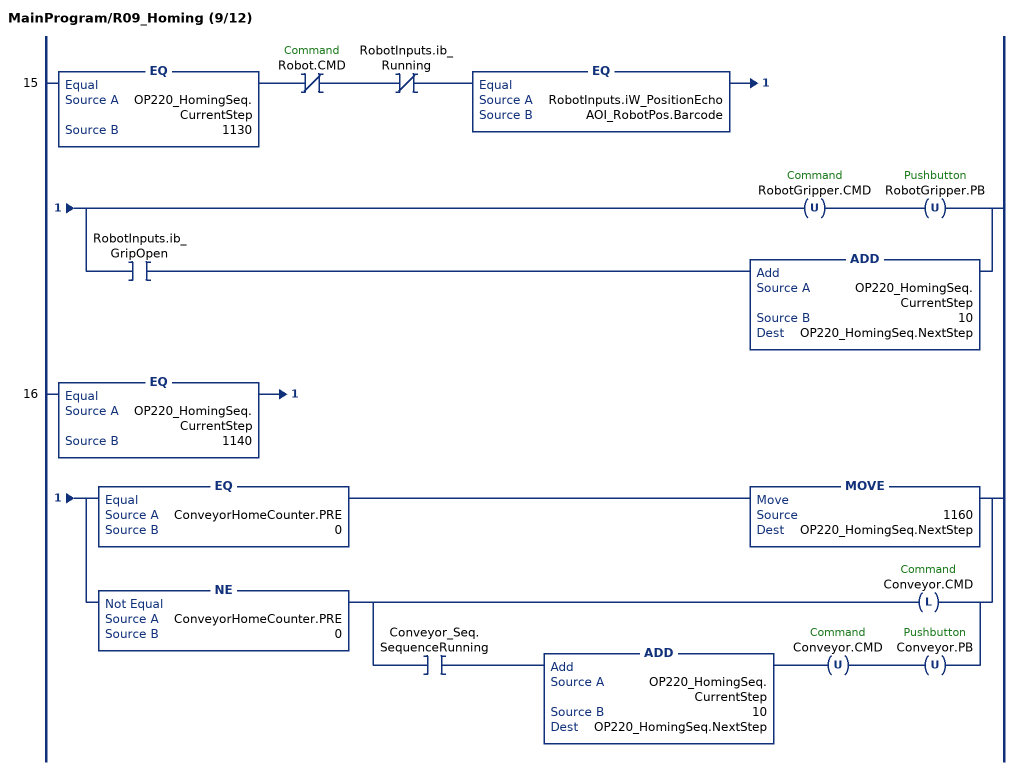
   15: EQ(OP220_HomingSeq.CurrentStep,1130)XIO(Robot.CMD)XIO(RobotInputs.ib_Running)EQ(RobotInputs.iW_PositionEcho,AOI_RobotPos.Barcode)[OTU(RobotGripper.CMD) OTU(RobotGripper.PB) ,XIC(RobotInputs.ib_GripOpen) ADD(OP220_HomingSeq.CurrentStep,10,OP220_HomingSeq.NextStep) ];
   16: EQ(OP220_HomingSeq.CurrentStep,1140)[EQ(ConveyorHomeCounter.PRE,0) MOVE(1160,OP220_HomingSeq.NextStep) ,NE(ConveyorHomeCounter.PRE,0) [OTL(Conveyor.CMD) ,XIC(Conveyor_Seq.SequenceRunning) ADD(OP220_HomingSeq.CurrentStep,10,OP220_HomingSeq.NextStep) OTU(Conveyor.CMD) OTU(Conveyor.PB) ] ];
